TYPE (* View rendering style *)
  (* Standard: 61499-1 *)
  (* Version 0.3, 2004-09-29, JHC, Rockwell Automation, Added PALLET. *)
  (* Version 0.2, 2002-05-21, JHC, Rockwell Automation, Deleted CLAMP. *)
  (* Version 0.1, 2002-04-25, JHC, Rockwell Automation, Added CLAMP, EMPTY; moved to fb.rt.mva. *)
  (* Version 0.0, 2002-04-01, JHC, Rockwell Automation *)
  (* Compiler header: package fb.rt.mva; *)
  (* Compiler Java Sun JDK 1.4.2 *)
  (* ASN.1 tag PRIVATE 21 *)
  VSTYLE : (
    BAR,
    SLIDER,
    CYLINDER,
    BALL,
    DISC,
    TOOL_OFF,
    TOOL_ON,
    SOLENOID,
    RING,
    PEG,
    PEGRING,
    EMPTY, (* Empty Box *)
    NONE,
    PALLET
  );
END_TYPE
